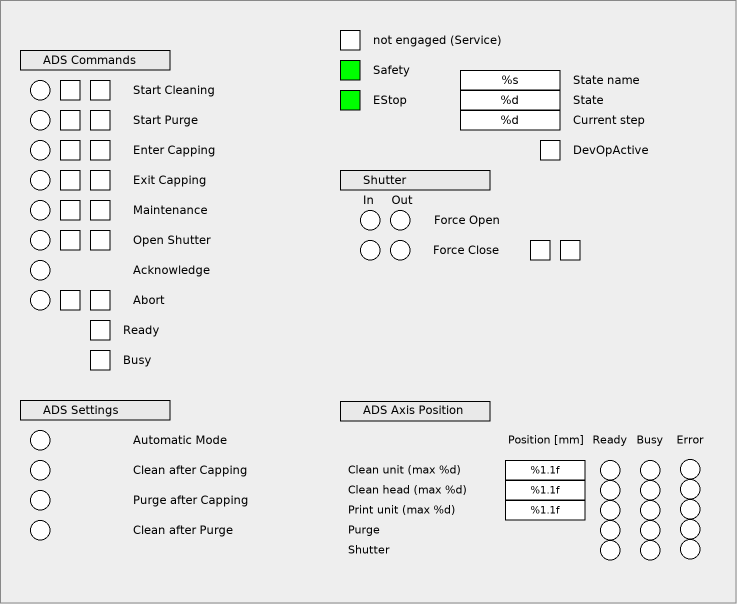
VISUALIZATION _VISU_CleanProcess  // 737x604
VAR_IN_OUT
  mInst            : FB_CleaningProcess;
  mInst_AdsProcess : FB_ADS_CleanProcess;
  mInst_AdsCU      : FB_ADS_CleanAxis;
  mInst_AdsCH      : FB_ADS_CleanAxis;
  mInst_AdsPU      : FB_ADS_CleanAxis;
  mInst_AdsPurge   : FB_ADS_CleanAxis;
  _bShutterExist   : BOOL;
  mInst_AdsShutter : FB_ADS_CleanAxis;
  mInst_FbShutter  : FB_SHUTTER;
END_VAR
    Rectangle (0,0 737x604)
    Polyline (20,50)
    Polyline (360,360)
    Rectangle (130,80 90x20), "Start Cleaning"
    Ellipse (30,80 20x20), colour toggle: mInst_AdsProcess.bI_Clean
        tap mInst_AdsProcess.bI_Clean
    Rectangle (130,110 90x20), "Start Purge"
    Rectangle (130,140 90x20), "Enter Capping"
    Rectangle (130,170 90x20), "Exit Capping"
    Rectangle (130,200 90x20), "Maintenance"
    RoundedRectangle (90,320 20x20), colour toggle: mInst_AdsProcess.bO_Ready
    Rectangle (120,320 120x20), "Ready"
    Rectangle (460,70 100x20), "%s", text variable: mInst.sL_CurrentState^.sL_StateName
    Rectangle (570,70 100x20), "State name"
    Rectangle (460,90 100x20), "%d", text variable: mInst.sL_CurrentState^.iL_State
    Rectangle (570,90 100x20), "State"
    Rectangle (20,50 150x20)
    Rectangle (40,50 130x20), "ADS Commands"
    RoundedRectangle (60,80 20x20), colour toggle: mInst_AdsProcess.bO_CleanCanEx
    RoundedRectangle (90,80 20x20), colour toggle: mInst_AdsProcess.bO_CleanExec
    Ellipse (30,110 20x20), colour toggle: mInst_AdsProcess.bI_Purge
        tap mInst_AdsProcess.bI_Purge
    RoundedRectangle (60,110 20x20), colour toggle: mInst_AdsProcess.bO_PurgeCanEx
    RoundedRectangle (90,110 20x20), colour toggle: mInst_AdsProcess.bO_PurgeExec
    Ellipse (30,140 20x20), colour toggle: mInst_AdsProcess.bI_StartCapping
        tap mInst_AdsProcess.bI_StartCapping
    RoundedRectangle (60,140 20x20), colour toggle: mInst_AdsProcess.bO_StartCappingCanEx
    RoundedRectangle (90,140 20x20), colour toggle: mInst_AdsProcess.bO_StartCappingExec
    Ellipse (30,170 20x20), colour toggle: mInst_AdsProcess.bI_StopCapping
        tap mInst_AdsProcess.bI_StopCapping
    RoundedRectangle (60,170 20x20), colour toggle: mInst_AdsProcess.bO_StopCappingCanEx
    RoundedRectangle (90,170 20x20), colour toggle: mInst_AdsProcess.bO_StopCappingExec
    Ellipse (30,200 20x20), colour toggle: mInst_AdsProcess.bI_Maintenance
        tap mInst_AdsProcess.bI_Maintenance
    RoundedRectangle (60,200 20x20), colour toggle: mInst_AdsProcess.bO_MaintenanceCanEx
    RoundedRectangle (90,200 20x20), colour toggle: mInst_AdsProcess.bO_MaintenanceExec
    Rectangle (130,290 90x20), "Abort"
    Ellipse (30,290 20x20), colour toggle: mInst_AdsProcess.bI_Abort
        tap mInst_AdsProcess.bI_Abort
    RoundedRectangle (60,290 20x20), colour toggle: mInst_AdsProcess.bO_AbortCanEx
    RoundedRectangle (90,290 20x20), colour toggle: mInst_AdsProcess.bO_AbortExec
    RoundedRectangle (90,350 20x20), colour toggle: mInst_AdsProcess.bO_Busy
    Rectangle (120,350 120x20), "Busy"
    Rectangle (20,400 150x20)
    Rectangle (40,400 130x20), "ADS Settings"
    Polyline (40,360)
    RoundedRectangle (340,90 20x20), colour toggle: mInst.bI_Emergency
    Rectangle (370,30 180x20), "not engaged (Service)"
    Rectangle (505,460 80x20), "%1.1f", text variable: mInst_AdsCU.sO_AxisPosition.fO_Val
    Rectangle (505,480 80x20), "%1.1f", text variable: mInst_AdsCH.sO_AxisPosition.fO_Val
    Rectangle (505,500 80x20), "%1.1f", text variable: mInst_AdsPU.sO_AxisPosition.fO_Val
    Ellipse (600,460 20x20), colour toggle: mInst_AdsCU.bO_Ready
    Ellipse (640,460 20x20), colour toggle: mInst_AdsCU.bO_Busy
    Ellipse (600,480 20x20), colour toggle: mInst_AdsCH.bO_Ready
    Ellipse (640,480 20x20), colour toggle: mInst_AdsCH.bO_Busy
    Ellipse (600,500 20x20), colour toggle: mInst_AdsPU.bO_Ready
    Ellipse (640,500 20x20), colour toggle: mInst_AdsPU.bO_Busy
    Rectangle (590,430 40x20), "Ready"
    Rectangle (630,430 40x20), "Busy"
    Rectangle (505,430 83x20), "Position [mm]"
    Rectangle (340,401 150x20)
    Rectangle (360,400 130x20), "ADS Axis Position"
    Ellipse (600,520 20x20), colour toggle: mInst_AdsPurge.bO_Ready
    Ellipse (640,520 20x20), colour toggle: mInst_AdsPurge.bO_Busy
    Rectangle (345,520 150x20), "Purge"
    Ellipse (680,459 20x20), colour toggle: mInst_AdsCU.bO_Error
        toggle mInst_AdsCU.bI_FaultAck
    Ellipse (680,479 20x20), colour toggle: mInst_AdsCH.bO_Error
        toggle mInst_AdsCH.bI_FaultAck
    Ellipse (680,499 20x20), colour toggle: mInst_AdsPU.bO_Error
        tap mInst_AdsPU.bI_FaultAck
    Rectangle (670,430 40x20), "Error"
    Ellipse (680,519 20x20), colour toggle: mInst_AdsPurge.bO_Error
    RoundedRectangle (340,60 20x20), colour toggle: NOT mInst.bI_SafetyOk
    RoundedRectangle (340,30 20x20), colour toggle: mInst.bI_UsrService
    Rectangle (370,60 80x20), "Safety"
    Rectangle (370,90 80x20), "EStop"
    Rectangle (345,460 150x20), "Clean unit (max %d)", text variable: mInst_AdsCU.sO_AxisPosition.fC_Max
    Rectangle (345,480 150x20), "Clean head (max %d)", text variable: mInst_AdsCH.sO_AxisPosition.fC_Max
    Rectangle (345,500 150x20), "Print unit (max %d)", text variable: mInst_AdsPU.sO_AxisPosition.fC_Max
    Rectangle (460,110 100x20), "%d", text variable: mInst.sL_CurrentState^.iL_CurrentStep
    Rectangle (570,110 100x20), "Current step"
    RoundedRectangle (540,140 20x20), colour toggle: mInst.sL_CurrentState^.bL_DevOpActive
    Rectangle (570,140 100x20), "DevOpActive"
    Rectangle (130,430 103x20), "Automatic Mode"
    Ellipse (30,430 20x20), colour toggle: mInst_AdsProcess.bI_AutoMode
        toggle mInst_AdsProcess.bI_AutoMode
    Rectangle (130,460 150x20), "Clean after Capping"
    Ellipse (30,460 20x20), colour toggle: mInst_AdsProcess.bI_CleanAfterCapp
        toggle mInst_AdsProcess.bI_CleanAfterCapp
    Rectangle (130,520 150x20), "Clean after Purge"
    Ellipse (30,520 20x20), colour toggle: mInst_AdsProcess.bI_CleanAfterPurge
        toggle mInst_AdsProcess.bI_CleanAfterPurge
    Rectangle (130,490 150x20), "Purge after Capping"
    Ellipse (30,490 20x20), colour toggle: mInst_AdsProcess.bI_PurgeAfterCapp
        toggle mInst_AdsProcess.bI_PurgeAfterCapp
    Rectangle (130,260 90x20), "Acknowledge"
    Ellipse (30,260 20x20), colour toggle: mInst_AdsProcess.bI_Maintenance
        tap mInst_AdsProcess.bI_AcknowledgeError
    Polyline (480,130), invisible if: NOT _bShutterExist
    Rectangle (431,210 81x20), "Force Open", invisible if: NOT _bShutterExist
    Ellipse (360,210 20x20), invisible if: NOT _bShutterExist
        toggle mInst_FbShutter.bI_ForceInletOpen
    Rectangle (430,240 82x20), "Force Close", invisible if: NOT _bShutterExist
    Ellipse (360,240 20x20), invisible if: NOT _bShutterExist
        toggle mInst_FbShutter.bI_ForceInletClose
    Rectangle (340,170 150x20), invisible if: NOT _bShutterExist
    Rectangle (360,170 130x20), "Shutter", invisible if: NOT _bShutterExist
    RoundedRectangle (530,240 20x20), colour toggle: mInst_FbShutter.bI_ShutterInletClosed, invisible if: NOT _bShutterExist
    Ellipse (390,210 20x20), invisible if: NOT _bShutterExist
        toggle mInst_FbShutter.bI_ForceOutletOpen
    Ellipse (390,240 20x20), invisible if: NOT _bShutterExist
        toggle mInst_FbShutter.bI_ForceOutletClose
    RoundedRectangle (560,240 20x20), colour toggle: mInst_FbShutter.bI_ShutterOutletClosed, invisible if: NOT _bShutterExist
    Rectangle (360,190 81x20), "In Out", invisible if: NOT _bShutterExist
    Rectangle (130,230 90x20), "Open Shutter", invisible if: NOT _bShutterExist
    Ellipse (30,230 20x20), invisible if: NOT _bShutterExist
        tap mInst_AdsProcess.bI_OpenShutter
    RoundedRectangle (60,230 20x20), colour toggle: mInst_AdsProcess.bO_OpenShutterCanEx, invisible if: NOT _bShutterExist
    RoundedRectangle (90,230 20x20), colour toggle: mInst_AdsProcess.bO_OpenShutterExec, invisible if: NOT _bShutterExist
    Ellipse (600,540 20x20), colour toggle: mInst_AdsShutter.bO_Ready, invisible if: NOT _bShutterExist
    Ellipse (640,540 20x20), colour toggle: mInst_AdsShutter.bO_Busy, invisible if: NOT _bShutterExist
    Rectangle (345,540 150x20), "Shutter", invisible if: NOT _bShutterExist
    Ellipse (680,539 20x20), colour toggle: mInst_AdsShutter.bO_Error, invisible if: NOT _bShutterExist
END_VISUALIZATION

(* stored: Version 1.1.0.1, ProductVersion 3.1.4024.11
   Visu _VISU_CleanProcess: Id {8578fc96-0785-4854-b88f-b29b1227eae5} *)
